// TIA Portal project "Gaugin station" (V16)

(* hardware
DEVICE "ET 200SP station_1"  ET 200SP-Station
   slot 0: "IO device_1"  IM 155-6 PN/2 HF  6ES7 155-6AU01-0CN0  V4.2
   slot 0: "Rack_0"  Rack  6ES5 710-8MAx1
   slot 1: "DI 8x24VDC HF_1"  DI 8x24VDC HF  6ES7 131-6BF00-0CA0  V2.0
      slot 1: "DI 8x24VDC HF_1"  DI 8x24VDC HF
   slot 2: "DI 8x24VDC HF_2"  DI 8x24VDC HF  6ES7 131-6BF00-0CA0  V2.0
      slot 1: "DI 8x24VDC HF_2"  DI 8x24VDC HF
   slot 3: "DI 8x24VDC HF_3"  DI 8x24VDC HF  6ES7 131-6BF00-0CA0  V2.0
      slot 1: "DI 8x24VDC HF_3"  DI 8x24VDC HF
   slot 4: "DQ 8x24VDC/0.5A HF_1"  DQ 8x24VDC/0.5A HF  6ES7 132-6BF00-0CA0  V2.0
      slot 1: "DQ 8x24VDC/0.5A HF_1"  DQ 8x24VDC/0.5A HF
   slot 5: "DQ 8x24VDC/0.5A HF_2"  DQ 8x24VDC/0.5A HF  6ES7 132-6BF00-0CA0  V2.0
      slot 1: "DQ 8x24VDC/0.5A HF_2"  DQ 8x24VDC/0.5A HF
   slot 6: "Server module_1"  Server module  6ES7 193-6PA00-0AA0  V1.1
      slot 1: "Server module_1"  Server module
   slot 127: "BA 2xRJ45"  BA 2xRJ45  6ES7 193-6AR00-0AA0  V0.0
      slot 1: "Port_1"  X1 P1 R  6ES7 193-6AR00-0AA0  V0.0
      slot 2: "Port_2"  X1 P2 R  6ES7 193-6AR00-0AA0  V0.0
DEVICE "S7-1200 station_1"  S7-1200 Station
   slot 0: "Rack_0"  S7-1200 Rack  Rack  V1.0
   slot 1: "PLC_1"  CPU 1214C DC/DC/DC  6ES7 214-1AG40-0XB0  V4.4
DEVICE "SCALANCE X005"  SCALANCE X-Station
   slot 0: "Switch_1"  6GK5 005-0BA00-1AB2  V1.0
   slot 0: "SCALANCE X rack"  Rail
*)

// ===== PLC "PLC_1"  CPU 1214C DC/DC/DC =====

VAR_GLOBAL   // PLC tag table "Default tag table"
   "Tag_1" AT %M98.0 : Bool;
   "Tag_2" AT %M98.1 : Bool;
   "Tag_3" AT %M98.2 : Bool;
   "Clock_Byte" AT %MB200 : Byte;
   "Clock_10Hz" AT %M200.0 : Bool;
   "Clock_5Hz" AT %M200.1 : Bool;
   "Clock_2.5Hz" AT %M200.2 : Bool;
   "Clock_2Hz" AT %M200.3 : Bool;
   "Clock_1.25Hz" AT %M200.4 : Bool;
   "Clock_1Hz" AT %M200.5 : Bool;
   "Clock_0.625Hz" AT %M200.6 : Bool;
   "Clock_0.5Hz" AT %M200.7 : Bool;
   "Tag_4" AT %M10.6 : Bool;
   "System_Byte" AT %MB30 : Byte;
   "FirstScan" AT %M30.0 : Bool;
   "DiagStatusUpdate" AT %M30.1 : Bool;
   "AlwaysTRUE" AT %M30.2 : Bool;
   "AlwaysFALSE" AT %M30.3 : Bool;
END_VAR

VAR_GLOBAL   // PLC tag table "IO_tags"
   "START BUTTON  (N.O.)" AT %I0.0 : Bool;
   "STOP BUTTON (N.C.)" AT %I0.1 : Bool;
   "EMERGENCY STOP BUTTON (N.C.)" AT %I0.2 : Bool;
   "OUTPUT POWER ON (WHITE)" AT %I0.3 : Bool;
   "INPUT 1 FROM PREVIOUS STATION" AT %I0.4 : Bool;
   "INPUT 2 FROM PREVIOUS STATION" AT %I0.5 : Bool;
   "INPUT 1 FROM NEXT STATION" AT %I0.6 : Bool;
   "INPUT 2 FROM NEXT STATION" AT %I0.7 : Bool;
   "RESET/AUTO SWITCH (RESET)" AT %I1.0 : Bool;
   "RESET/AUTO SWITCH (AUTO)" AT %I1.1 : Bool;
   "REJECT CYLINDER 3A RETRACTED" AT %I1.2 : Bool;
   "REJECT CYLINDER 3A EXTENDED" AT %I1.3 : Bool;
   "TRANSFER CYLINDER 1A RETRACTED" AT %I1.4 : Bool;
   "TRANSFER CYLINDER 1A EXTENDED" AT %I1.5 : Bool;
   "TRAVERSE IN END OF TRAVEL POSITION" AT %I4.6 : Bool;
   "TRAVERSE IN START OF TRAVEL POSITION" AT %I4.7 : Bool;
   "PART IN HEIGHT MEASURING POSITION (INDUCTIVE SENSOR)" AT %I2.0 : Bool;
   "PART HEIGHT READING (ULTRASONIC SENSOR)" AT %I2.1 : Bool;
   "PORT NOT DETECTED (LIGHT SENSOR)" AT %I2.2 : Bool;
   "AUTOMATIC ON  LAMP (GREEN)" AT %Q0.0 : Bool;
   "OUTPUT 1 TO PREVIOUS STATION" AT %Q0.1 : Bool;
   "OUTPUT 2 TO PREVIOUS STATION" AT %Q0.2 : Bool;
   "OUTPUT 1 TO NEXT STATION" AT %Q0.3 : Bool;
   "OUTPUT 2 TO NEXT STATION" AT %Q0.4 : Bool;
   "EXTEND REJECT CYLINDER" AT %Q0.5 : Bool;
   "EXTEND TRANSFER CYLINDER" AT %Q0.6 : Bool;
   "RETRACT TRANSFER CYLINDER" AT %Q0.7 : Bool;
   "MOTOR STARTER FORWARD" AT %Q1.0 : Bool;
   "MOTOR STARTER REVERSE" AT %Q1.1 : Bool;
   "EXTEND LIFT CYLINDER" AT %Q3.1 : Bool;
END_VAR

DATA_BLOCK "Modes Data"   // DB1
{ S7_Optimized_Access := 'TRUE' }
VERSION : 0.1
   VAR
      Automatic : Bool;
      Manual : Bool;
      Reset : Bool;
      "Pre-Automatic" : Bool;
   END_VAR
BEGIN
END_DATA_BLOCK

DATA_BLOCK "Outputs Data"   // DB2
{ S7_Optimized_Access := 'TRUE' }
VERSION : 0.1
   VAR
      "Extend reject cylinder" : Bool;
      "Extend transfer cylinder" : Bool;
      "Retract transfer cylinder" : Bool;
      "Motor forward" : Bool;
      "Motor Reverse" : Bool;
      "Extend Lift Cylinder" : Bool;
      Output : Bool;
   END_VAR
BEGIN
END_DATA_BLOCK

DATA_BLOCK "status data"   // DB3
{ S7_Optimized_Access := 'TRUE' }
VERSION : 0.1
   VAR
      steps : Int;
      "port not detected" : Bool;
      "height detected" : Bool;
      next_step : Bool;
      input_from_previous_Station : Bool;
   END_VAR
BEGIN
END_DATA_BLOCK

// folder: System blocks/Program resources

DATA_BLOCK "port_detection_wait"   // DB4
{ S7_Optimized_Access := 'TRUE' }
AUTHOR : Simatic
FAMILY : IEC
NAME : IEC_TMR
VERSION : 1.0
// stored: InstanceOfName IEC_TIMER
"IEC_TIMER"
BEGIN
END_DATA_BLOCK

DATA_BLOCK "retract_delay"   // DB5
{ S7_Optimized_Access := 'TRUE' }
AUTHOR : Simatic
FAMILY : IEC
NAME : IEC_TMR
VERSION : 1.0
// stored: InstanceOfName IEC_TIMER
"IEC_TIMER"
BEGIN
END_DATA_BLOCK

DATA_BLOCK "next_step_delay"   // DB6
{ S7_Optimized_Access := 'TRUE' }
AUTHOR : Simatic
FAMILY : IEC
NAME : IEC_TMR
VERSION : 1.0
// stored: InstanceOfName IEC_TIMER
"IEC_TIMER"
BEGIN
END_DATA_BLOCK

DATA_BLOCK "height_Timer_0_DB"   // DB7
{ S7_Optimized_Access := 'TRUE' }
AUTHOR : Simatic
FAMILY : IEC
NAME : IEC_TMR
VERSION : 1.0
// stored: InstanceOfName IEC_TIMER
"IEC_TIMER"
BEGIN
END_DATA_BLOCK

DATA_BLOCK "retract_wait"   // DB8
{ S7_Optimized_Access := 'TRUE' }
AUTHOR : Simatic
FAMILY : IEC
NAME : IEC_TMR
VERSION : 1.0
// stored: InstanceOfName IEC_TIMER
"IEC_TIMER"
BEGIN
END_DATA_BLOCK

DATA_BLOCK "next_step_wait_1"   // DB9
{ S7_Optimized_Access := 'TRUE' }
AUTHOR : Simatic
FAMILY : IEC
NAME : IEC_TMR
VERSION : 1.0
// stored: InstanceOfName IEC_TIMER
"IEC_TIMER"
BEGIN
END_DATA_BLOCK

DATA_BLOCK "motor_wait"   // DB10
{ S7_Optimized_Access := 'TRUE' }
AUTHOR : Simatic
FAMILY : IEC
NAME : IEC_TMR
VERSION : 1.0
// stored: InstanceOfName IEC_TIMER
"IEC_TIMER"
BEGIN
END_DATA_BLOCK

DATA_BLOCK "extend_retract_wait"   // DB11
{ S7_Optimized_Access := 'TRUE' }
AUTHOR : Simatic
FAMILY : IEC
NAME : IEC_TMR
VERSION : 1.0
// stored: InstanceOfName IEC_TIMER
"IEC_TIMER"
BEGIN
END_DATA_BLOCK

// folder: (top level)

FUNCTION "Modes" : Void   // FC1, LAD
TITLE = Modes Setup
{ S7_Optimized_Access := 'TRUE' }
VERSION : 0.1
BEGIN

REGION Network 1: Automatic Mode
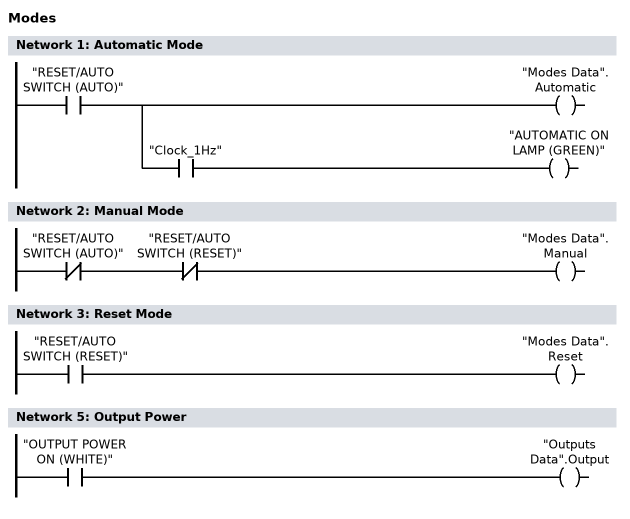
   RUNG wire#powerrail
      Contact( "RESET/AUTO SWITCH (AUTO)" )
      wire#w1
      Coil( "Modes Data".Automatic )
   END_RUNG
   RUNG wire#w1
      Contact( "Clock_1Hz" )
      Coil( "AUTOMATIC ON  LAMP (GREEN)" )
   END_RUNG
   // the same network as SCL:
   "Modes Data".Automatic := "RESET/AUTO SWITCH (AUTO)";
   "AUTOMATIC ON  LAMP (GREEN)" := "RESET/AUTO SWITCH (AUTO)" AND "Clock_1Hz";
END_REGION

REGION Network 2: Manual Mode
   RUNG wire#powerrail
      I_Contact( "RESET/AUTO SWITCH (AUTO)" )
      I_Contact( "RESET/AUTO SWITCH (RESET)" )
      Coil( "Modes Data".Manual )
   END_RUNG
   // the same network as SCL:
   "Modes Data".Manual := NOT "RESET/AUTO SWITCH (AUTO)" AND NOT "RESET/AUTO SWITCH (RESET)";
END_REGION

REGION Network 3: Reset Mode
   RUNG wire#powerrail
      Contact( "RESET/AUTO SWITCH (RESET)" )
      Coil( "Modes Data".Reset )
   END_RUNG
   // the same network as SCL:
   "Modes Data".Reset := "RESET/AUTO SWITCH (RESET)";
END_REGION

REGION Network 4: Pre-Automatic Mode
END_REGION

REGION Network 5: Output Power
   RUNG wire#powerrail
      Contact( "OUTPUT POWER ON (WHITE)" )
      Coil( "Outputs Data".Output )
   END_RUNG
   // the same network as SCL:
   "Outputs Data".Output := "OUTPUT POWER ON (WHITE)";
END_REGION
END_FUNCTION

FUNCTION "Outputs" : Void   // FC2, LAD
{ S7_Optimized_Access := 'TRUE' }
VERSION : 0.1
BEGIN

REGION Network 1: Reject Cylinder
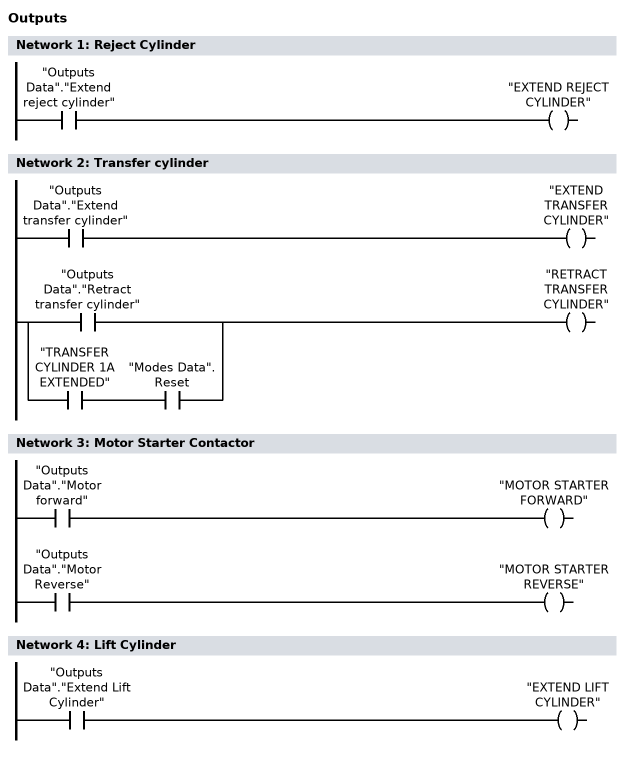
   RUNG wire#powerrail
      Contact( "Outputs Data"."Extend reject cylinder" )
      Coil( "EXTEND REJECT CYLINDER" )
   END_RUNG
   // the same network as SCL:
   "EXTEND REJECT CYLINDER" := "Outputs Data"."Extend reject cylinder";
END_REGION

REGION Network 2: Transfer cylinder
   RUNG wire#powerrail
      Contact( "Outputs Data"."Extend transfer cylinder" )
      Coil( "EXTEND TRANSFER CYLINDER" )
   END_RUNG
   RUNG wire#powerrail
      Contact( "Outputs Data"."Retract transfer cylinder" )
      wire#w1
      Coil( "RETRACT TRANSFER CYLINDER" )
   END_RUNG
   RUNG wire#powerrail
      Contact( "TRANSFER CYLINDER 1A EXTENDED" )
      Contact( "Modes Data".Reset )
   END_RUNG wire#w1
   // the same network as SCL:
   "EXTEND TRANSFER CYLINDER" := "Outputs Data"."Extend transfer cylinder";
   "RETRACT TRANSFER CYLINDER" := "Outputs Data"."Retract transfer cylinder" OR ("TRANSFER CYLINDER 1A EXTENDED" AND "Modes Data".Reset);
END_REGION

REGION Network 3: Motor Starter Contactor
   RUNG wire#powerrail
      Contact( "Outputs Data"."Motor forward" )
      Coil( "MOTOR STARTER FORWARD" )
   END_RUNG
   RUNG wire#powerrail
      Contact( "Outputs Data"."Motor Reverse" )
      Coil( "MOTOR STARTER REVERSE" )
   END_RUNG
   // the same network as SCL:
   "MOTOR STARTER FORWARD" := "Outputs Data"."Motor forward";
   "MOTOR STARTER REVERSE" := "Outputs Data"."Motor Reverse";
END_REGION

REGION Network 4: Lift Cylinder
   RUNG wire#powerrail
      Contact( "Outputs Data"."Extend Lift Cylinder" )
      Coil( "EXTEND LIFT CYLINDER" )
   END_RUNG
   // the same network as SCL:
   "EXTEND LIFT CYLINDER" := "Outputs Data"."Extend Lift Cylinder";
END_REGION
END_FUNCTION

FUNCTION "operation" : Void   // FC4, LAD
{ S7_Optimized_Access := 'TRUE' }
VERSION : 0.1
   VAR_TEMP   // added for the SCL form of the ladder/FBD networks
      _w1 : Bool;
   END_VAR
BEGIN

REGION Network 1
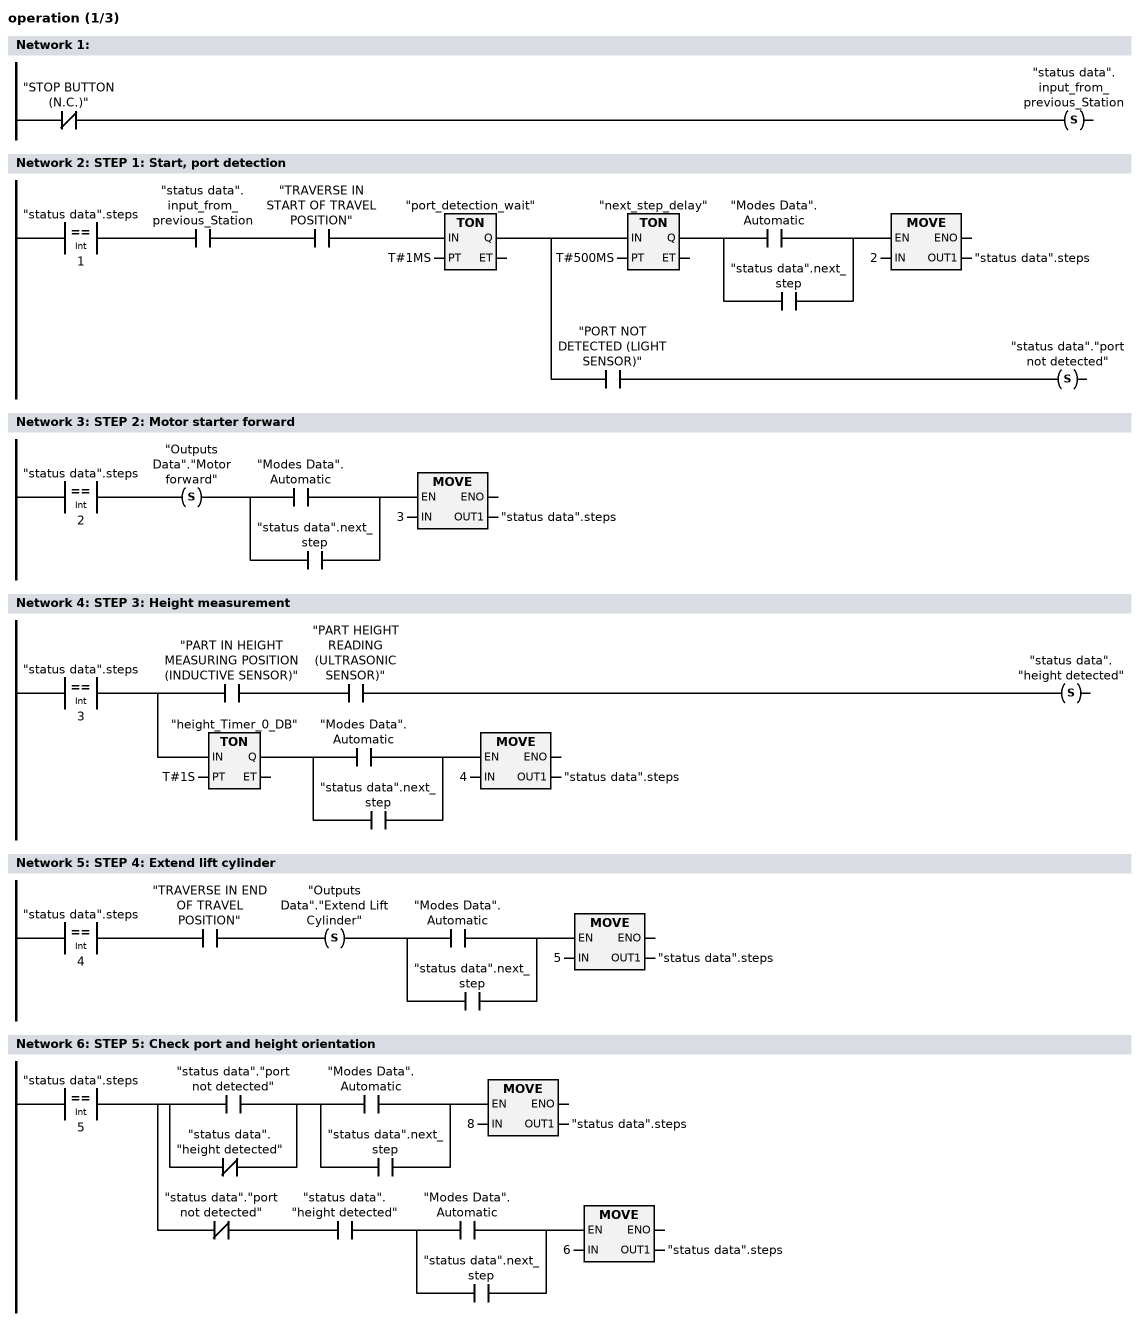
   RUNG wire#powerrail
      I_Contact( "STOP BUTTON (N.C.)" )
      S_Coil( "status data".input_from_previous_Station )
   END_RUNG
   // the same network as SCL:
   IF NOT "STOP BUTTON (N.C.)" THEN "status data".input_from_previous_Station := TRUE; END_IF;
END_REGION

REGION Network 2: STEP 1: Start, port detection
   "port_detection_wait".TON(IN := ("status data".steps = 1) AND "status data".input_from_previous_Station AND "TRAVERSE IN START OF TRAVEL POSITION",
                           PT := T#1MS);
   "next_step_delay".TON(IN := "port_detection_wait".Q, PT := T#500MS);
   IF "next_step_delay".Q AND ("Modes Data".Automatic OR "status data".next_step) THEN
       "status data".steps := 2;
   END_IF;
   IF "port_detection_wait".Q AND "PORT NOT DETECTED (LIGHT SENSOR)" THEN
       "status data"."port not detected" := TRUE;
   END_IF;
END_REGION

REGION Network 3: STEP 2: Motor starter forward
   RUNG wire#powerrail
      { S7_Templates := "SrcType := Int" } EQ_Contact(in1 := "status data".steps, in2 := 2)
      S_Coil( "Outputs Data"."Motor forward" )
      wire#w1
      Contact( "Modes Data".Automatic )
      wire#w2
      Move(in := 3, out1 => "status data".steps)
   END_RUNG
   RUNG wire#w1
      Contact( "status data".next_step )
   END_RUNG wire#w2
   // the same network as SCL:
   #_w1 := "status data".steps = 2;
   IF #_w1 THEN "Outputs Data"."Motor forward" := TRUE; END_IF;
   IF #_w1 AND ("Modes Data".Automatic OR "status data".next_step) THEN "status data".steps := 3; END_IF;
END_REGION

REGION Network 4: STEP 3: Height measurement
   #_w1 := "status data".steps = 3;
   IF #_w1 AND "PART IN HEIGHT MEASURING POSITION (INDUCTIVE SENSOR)" AND "PART HEIGHT READING (ULTRASONIC SENSOR)" THEN
       "status data"."height detected" := TRUE;
   END_IF;
   "height_Timer_0_DB".TON(IN := #_w1, PT := T#1S);
   IF "height_Timer_0_DB".Q AND ("Modes Data".Automatic OR "status data".next_step) THEN
       "status data".steps := 4;
   END_IF;
END_REGION

REGION Network 5: STEP 4: Extend lift cylinder
   RUNG wire#powerrail
      { S7_Templates := "SrcType := Int" } EQ_Contact(in1 := "status data".steps, in2 := 4)
      Contact( "TRAVERSE IN END OF TRAVEL POSITION" )
      S_Coil( "Outputs Data"."Extend Lift Cylinder" )
      wire#w1
      Contact( "Modes Data".Automatic )
      wire#w2
      Move(in := 5, out1 => "status data".steps)
   END_RUNG
   RUNG wire#w1
      Contact( "status data".next_step )
   END_RUNG wire#w2
   // the same network as SCL:
   #_w1 := ("status data".steps = 4) AND "TRAVERSE IN END OF TRAVEL POSITION";
   IF #_w1 THEN "Outputs Data"."Extend Lift Cylinder" := TRUE; END_IF;
   IF #_w1 AND ("Modes Data".Automatic OR "status data".next_step) THEN "status data".steps := 5; END_IF;
END_REGION

REGION Network 6: STEP 5: Check port and height orientation
   RUNG wire#powerrail
      { S7_Templates := "SrcType := Int" } EQ_Contact(in1 := "status data".steps, in2 := 5)
      wire#w1
      Contact( "status data"."port not detected" )
      wire#w2
      Contact( "Modes Data".Automatic )
      wire#w3
      Move(in := 8, out1 => "status data".steps)
   END_RUNG
   RUNG wire#w1
      I_Contact( "status data"."height detected" )
   END_RUNG wire#w2
   RUNG wire#w2
      Contact( "status data".next_step )
   END_RUNG wire#w3
   RUNG wire#w1
      I_Contact( "status data"."port not detected" )
      Contact( "status data"."height detected" )
      wire#w4
      Contact( "Modes Data".Automatic )
      wire#w5
      Move(in := 6, out1 => "status data".steps)
   END_RUNG
   RUNG wire#w4
      Contact( "status data".next_step )
   END_RUNG wire#w5
   // the same network as SCL:
   #_w1 := "status data".steps = 5;
   IF #_w1 AND ("status data"."port not detected" OR NOT "status data"."height detected") AND ("Modes Data".Automatic OR "status data".next_step) THEN
       "status data".steps := 8;
   END_IF;
   IF #_w1 AND NOT "status data"."port not detected" AND "status data"."height detected" AND ("Modes Data".Automatic OR "status data".next_step) THEN
       "status data".steps := 6;
   END_IF;
END_REGION

REGION Network 7: STEP 6: Extend transfer cylinder
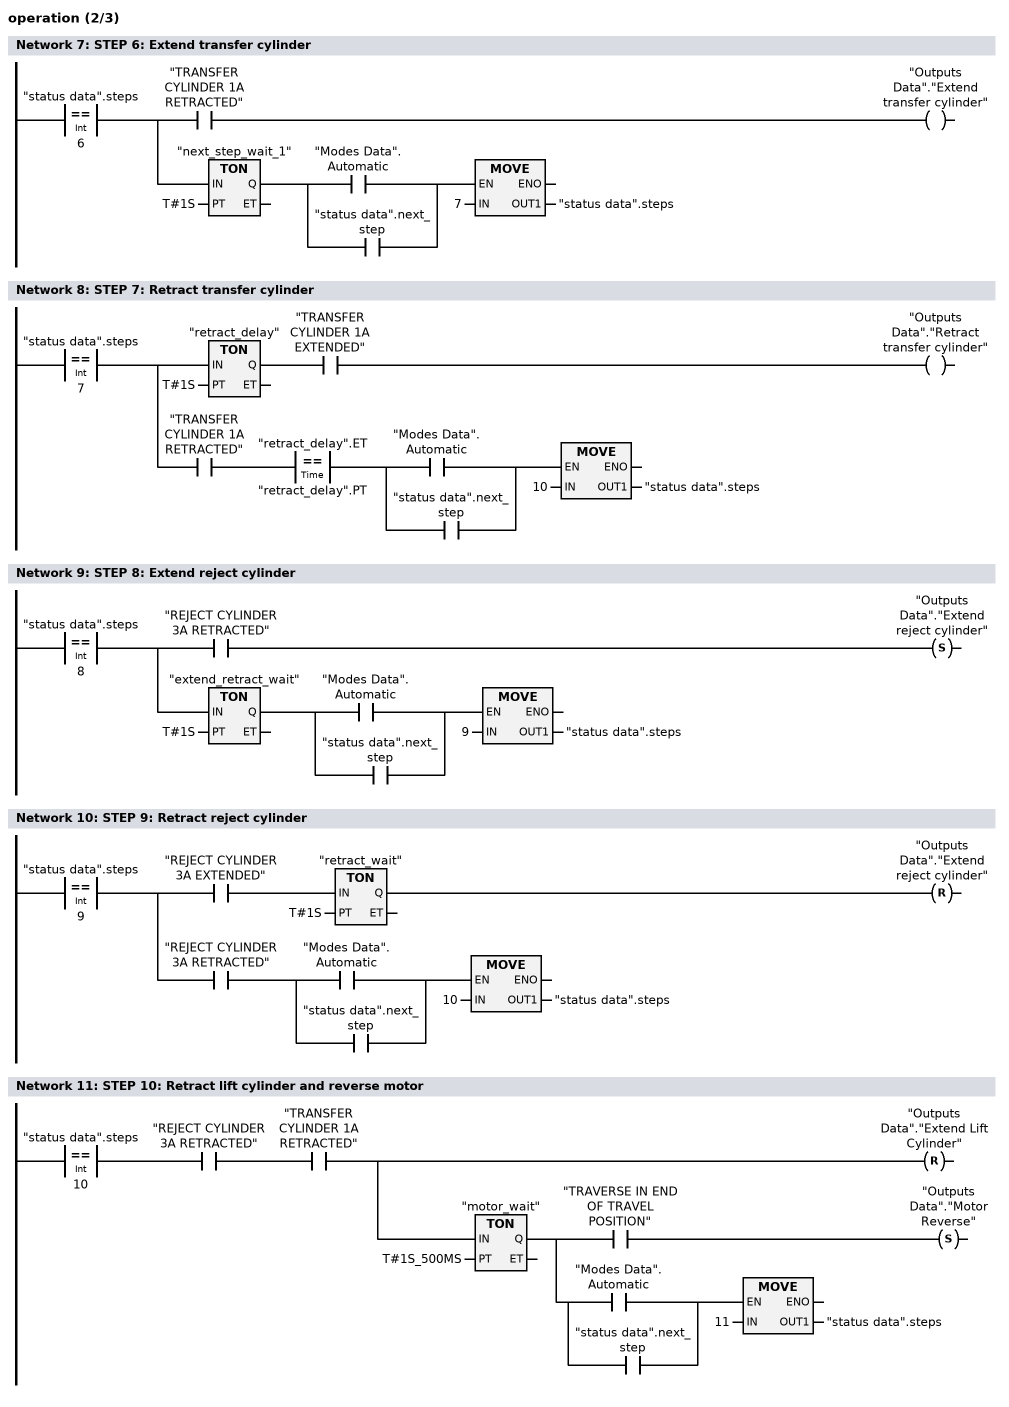
   #_w1 := "status data".steps = 6;
   "Outputs Data"."Extend transfer cylinder" := #_w1 AND "TRANSFER CYLINDER 1A RETRACTED";
   "next_step_wait_1".TON(IN := #_w1, PT := T#1S);
   IF "next_step_wait_1".Q AND ("Modes Data".Automatic OR "status data".next_step) THEN
       "status data".steps := 7;
   END_IF;
END_REGION

REGION Network 8: STEP 7: Retract transfer cylinder
   #_w1 := "status data".steps = 7;
   "retract_delay".TON(IN := #_w1, PT := T#1S);
   "Outputs Data"."Retract transfer cylinder" := "retract_delay".Q AND "TRANSFER CYLINDER 1A EXTENDED";
   IF #_w1 AND "TRANSFER CYLINDER 1A RETRACTED" AND ("retract_delay".ET = "retract_delay".PT) AND ("Modes Data".Automatic OR "status data".next_step) THEN
       "status data".steps := 10;
   END_IF;
END_REGION

REGION Network 9: STEP 8: Extend reject cylinder
   #_w1 := "status data".steps = 8;
   IF #_w1 AND "REJECT CYLINDER 3A RETRACTED" THEN "Outputs Data"."Extend reject cylinder" := TRUE; END_IF;
   "extend_retract_wait".TON(IN := #_w1, PT := T#1S);
   IF "extend_retract_wait".Q AND ("Modes Data".Automatic OR "status data".next_step) THEN
       "status data".steps := 9;
   END_IF;
END_REGION

REGION Network 10: STEP 9: Retract reject cylinder
   #_w1 := "status data".steps = 9;
   "retract_wait".TON(IN := #_w1 AND "REJECT CYLINDER 3A EXTENDED", PT := T#1S);
   IF "retract_wait".Q THEN "Outputs Data"."Extend reject cylinder" := FALSE; END_IF;
   IF #_w1 AND "REJECT CYLINDER 3A RETRACTED" AND ("Modes Data".Automatic OR "status data".next_step) THEN
       "status data".steps := 10;
   END_IF;
END_REGION

REGION Network 11: STEP 10: Retract lift cylinder and reverse motor
   #_w1 := ("status data".steps = 10) AND "REJECT CYLINDER 3A RETRACTED" AND "TRANSFER CYLINDER 1A RETRACTED";
   IF #_w1 THEN "Outputs Data"."Extend Lift Cylinder" := FALSE; END_IF;
   "motor_wait".TON(IN := #_w1, PT := T#1S_500MS);
   IF "motor_wait".Q AND "TRAVERSE IN END OF TRAVEL POSITION" THEN
       "Outputs Data"."Motor Reverse" := TRUE;
   END_IF;
   IF "motor_wait".Q AND ("Modes Data".Automatic OR "status data".next_step) THEN
       "status data".steps := 11;
   END_IF;
END_REGION

REGION Network 12: STEP 11: Reset to step 1
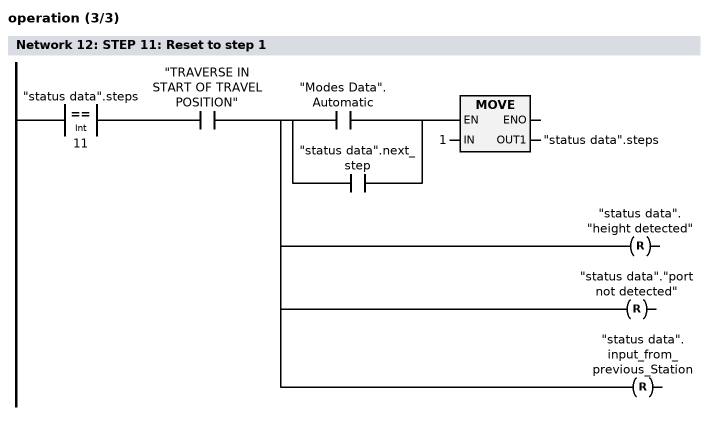
   RUNG wire#powerrail
      { S7_Templates := "SrcType := Int" } EQ_Contact(in1 := "status data".steps, in2 := 11)
      Contact( "TRAVERSE IN START OF TRAVEL POSITION" )
      wire#w1
      Contact( "Modes Data".Automatic )
      wire#w2
      Move(in := 1, out1 => "status data".steps)
   END_RUNG
   RUNG wire#w1
      Contact( "status data".next_step )
   END_RUNG wire#w2
   RUNG wire#w1
      R_Coil( "status data"."height detected" )
   END_RUNG
   RUNG wire#w1
      R_Coil( "status data"."port not detected" )
   END_RUNG
   RUNG wire#w1
      R_Coil( "status data".input_from_previous_Station )
   END_RUNG
   // the same network as SCL:
   #_w1 := ("status data".steps = 11) AND "TRAVERSE IN START OF TRAVEL POSITION";
   IF #_w1 AND ("Modes Data".Automatic OR "status data".next_step) THEN "status data".steps := 1; END_IF;
   IF #_w1 THEN
       "status data"."height detected" := FALSE;
       "status data"."port not detected" := FALSE;
       "status data".input_from_previous_Station := FALSE;
   END_IF;
END_REGION
END_FUNCTION

ORGANIZATION_BLOCK "Main"   // OB1, LAD, ProgramCycle
TITLE = "Main Program Sweep (Cycle)"
{ S7_Optimized_Access := 'TRUE' }
VERSION : 0.1
   VAR_INPUT
      Initial_Call : Bool;   // Initial call of this OB
      Remanence : Bool;   // =True, if remanent data are available
   END_VAR
   VAR_TEMP   // added for the SCL form of the ladder/FBD networks
      _w1 : Bool;
      _w2 : Bool;
   END_VAR
BEGIN

REGION Network 1: SETUP: output, start, reset
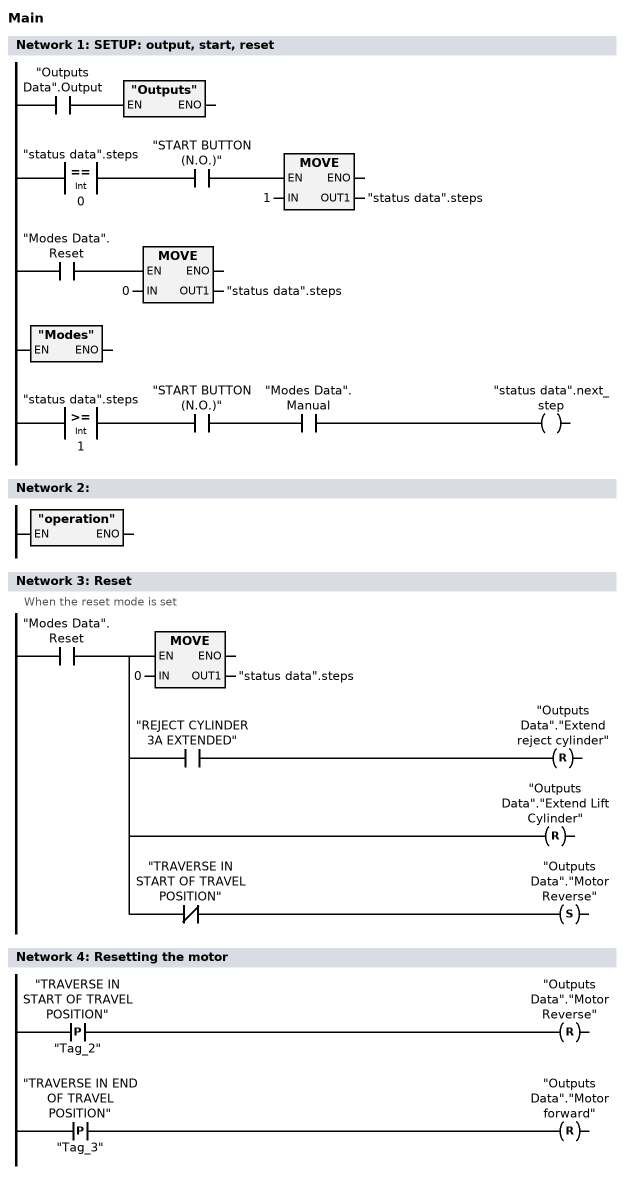
   RUNG wire#powerrail
      Contact( "Outputs Data".Output )
      "Outputs"()
   END_RUNG
   RUNG wire#powerrail
      { S7_Templates := "SrcType := Int" } EQ_Contact(in1 := "status data".steps, in2 := 0)
      Contact( "START BUTTON  (N.O.)" )
      Move(in := 1, out1 => "status data".steps)
   END_RUNG
   RUNG wire#powerrail
      Contact( "Modes Data".Reset )
      Move(in := 0, out1 => "status data".steps)
   END_RUNG
   RUNG wire#powerrail
      "Modes"()
   END_RUNG
   RUNG wire#powerrail
      { S7_Templates := "SrcType := Int" } GE_Contact(in1 := "status data".steps, in2 := 1)
      Contact( "START BUTTON  (N.O.)" )
      Contact( "Modes Data".Manual )
      Coil( "status data".next_step )
   END_RUNG
   // the same network as SCL:
   IF "Outputs Data".Output THEN "Outputs"(); END_IF;
   IF ("status data".steps = 0) AND "START BUTTON  (N.O.)" THEN "status data".steps := 1; END_IF;
   IF "Modes Data".Reset THEN "status data".steps := 0; END_IF;
   "Modes"();
   "status data".next_step := ("status data".steps >= 1) AND "START BUTTON  (N.O.)" AND "Modes Data".Manual;
END_REGION

REGION Network 2
   RUNG wire#powerrail
      "operation"()
   END_RUNG
   // the same network as SCL:
   "operation"();
END_REGION

REGION Network 3: Reset
   // When the reset mode is set
   RUNG wire#powerrail
      Contact( "Modes Data".Reset )
      wire#w1
      Move(in := 0, out1 => "status data".steps)
   END_RUNG
   RUNG wire#w1
      Contact( "REJECT CYLINDER 3A EXTENDED" )
      R_Coil( "Outputs Data"."Extend reject cylinder" )
   END_RUNG
   RUNG wire#w1
      R_Coil( "Outputs Data"."Extend Lift Cylinder" )
   END_RUNG
   RUNG wire#w1
      I_Contact( "TRAVERSE IN START OF TRAVEL POSITION" )
      S_Coil( "Outputs Data"."Motor Reverse" )
   END_RUNG
   // the same network as SCL:
   IF "Modes Data".Reset THEN "status data".steps := 0; END_IF;
   IF "Modes Data".Reset AND "REJECT CYLINDER 3A EXTENDED" THEN
       "Outputs Data"."Extend reject cylinder" := FALSE;
   END_IF;
   IF "Modes Data".Reset THEN "Outputs Data"."Extend Lift Cylinder" := FALSE; END_IF;
   IF "Modes Data".Reset AND NOT "TRAVERSE IN START OF TRAVEL POSITION" THEN
       "Outputs Data"."Motor Reverse" := TRUE;
   END_IF;
END_REGION

REGION Network 4: Resetting the motor
   RUNG wire#powerrail
      P_Contact(operand := "TRAVERSE IN START OF TRAVEL POSITION", bit := "Tag_2")
      R_Coil( "Outputs Data"."Motor Reverse" )
   END_RUNG
   RUNG wire#powerrail
      P_Contact(operand := "TRAVERSE IN END OF TRAVEL POSITION", bit := "Tag_3")
      R_Coil( "Outputs Data"."Motor forward" )
   END_RUNG
   // the same network as SCL:
   #_w1 := "TRAVERSE IN START OF TRAVEL POSITION" AND NOT "Tag_2";   // rising edge of "TRAVERSE IN START OF TRAVEL POSITION"
   "Tag_2" := "TRAVERSE IN START OF TRAVEL POSITION";
   IF #_w1 THEN "Outputs Data"."Motor Reverse" := FALSE; END_IF;
   #_w2 := "TRAVERSE IN END OF TRAVEL POSITION" AND NOT "Tag_3";   // rising edge of "TRAVERSE IN END OF TRAVEL POSITION"
   "Tag_3" := "TRAVERSE IN END OF TRAVEL POSITION";
   IF #_w2 THEN "Outputs Data"."Motor forward" := FALSE; END_IF;
END_REGION
END_ORGANIZATION_BLOCK